Yaskawa INFORM job: 3-Z.JBI

/JOB
//NAME 3-Z
///FOLDERNAME INNE
//POS
///NPOS 2,2,0,0,0,0
///TOOL 0
///POSTYPE PULSE
///PULSE
C00000=-1083,-6112,109948,-717,38573,314
C00001=-2374,-194541,-115082,-830,80221,-289
BC00000=277960,1059793,981056
BC00001=277960,1059793,283232
//INST
///DATE 2023/10/04 15:13
///ATTR SC,RW
///GROUP1 RB1,BS1
NOP
MOVJ C00000 BC00000 VJ=0.78
MOVJ C00001 BC00001 VJ=0.78
END
